// TIA Portal V17 export
// export: Created 2023-02-14T02:49:25.0894814Z, ExportSetting WithDefaults, DisplayName Totally Integrated Automation Portal, DisplayVersion V17, DisplayName TIA Portal Openness, DisplayVersion V17, DisplayName TIA Portal Teamcenter Gateway, DisplayVersion V17, DisplayName TIA Portal Version Control Interface, DisplayVersion V17, DisplayName SINAMICS Startdrive Advanced, DisplayVersion V17, DisplayName SINAMICS Startdrive G130, G150, S120, S150, SINAMICS MV, S210, DisplayVersion V17, DisplayName SINAMICS Startdrive G110M, G120, G120C, G120D, G120P, G115D, DisplayVersion V17, DisplayName STEP 7 Professional, DisplayVersion V17, DisplayName STEP 7 Safety, DisplayVersion V17, DisplayName WinCC Professional, DisplayVersion V17
FUNCTION_BLOCK "IO Analog Blending"   // FB10, LAD
{ S7_Optimized_Access := 'FALSE' }
VERSION : 0.1
// stored: AutoNumber true, IsIECCheckEnabled false, SetENOAutomatically false, UDAEnableTagReadback false
   VAR_INPUT
      Init : Bool;
      Reset : Bool;
   END_VAR
   VAR
      "LT-20.01" { S7_SetPoint := 'True'} : "Ana_w_K1K2";
      "LT-21.01" { S7_SetPoint := 'True'} : "Ana_w_K1K2";
      "LT-22.01" { S7_SetPoint := 'True'} : "Ana_w_K1K2";
      "LT-30.01" { S7_SetPoint := 'True'} : "Ana_w_K1K2";
      "LT-31.01" { S7_SetPoint := 'True'} : "Ana_w_K1K2";
      "LT-32.01" { S7_SetPoint := 'True'} : "Ana_w_K1K2";
      "FT-15.01" { S7_SetPoint := 'True'} : "Ana_w_K1K2";
      "FT-15.01Com" { S7_SetPoint := 'True'} : "Read FT Comm";
      "FT-22.01" { S7_SetPoint := 'True'} : "Ana_w_K1K2";
      "FT-22.01Com" { S7_SetPoint := 'True'} : "Read FT Comm";
      "FT-32.01" { S7_SetPoint := 'True'} : "Ana_w_K1K2";
      "FT-32.01Com" { S7_SetPoint := 'True'} : "Read FT Comm";
      "LT-40.01" { S7_SetPoint := 'True'} : "Ana_w_K1K2";
      "LT-41.01" { S7_SetPoint := 'True'} : "Ana_w_K1K2";
      "FT-00.01" { S7_SetPoint := 'True'} : "Ana_w_K1K2";
   END_VAR
BEGIN

REGION Network 1: LT-20.01
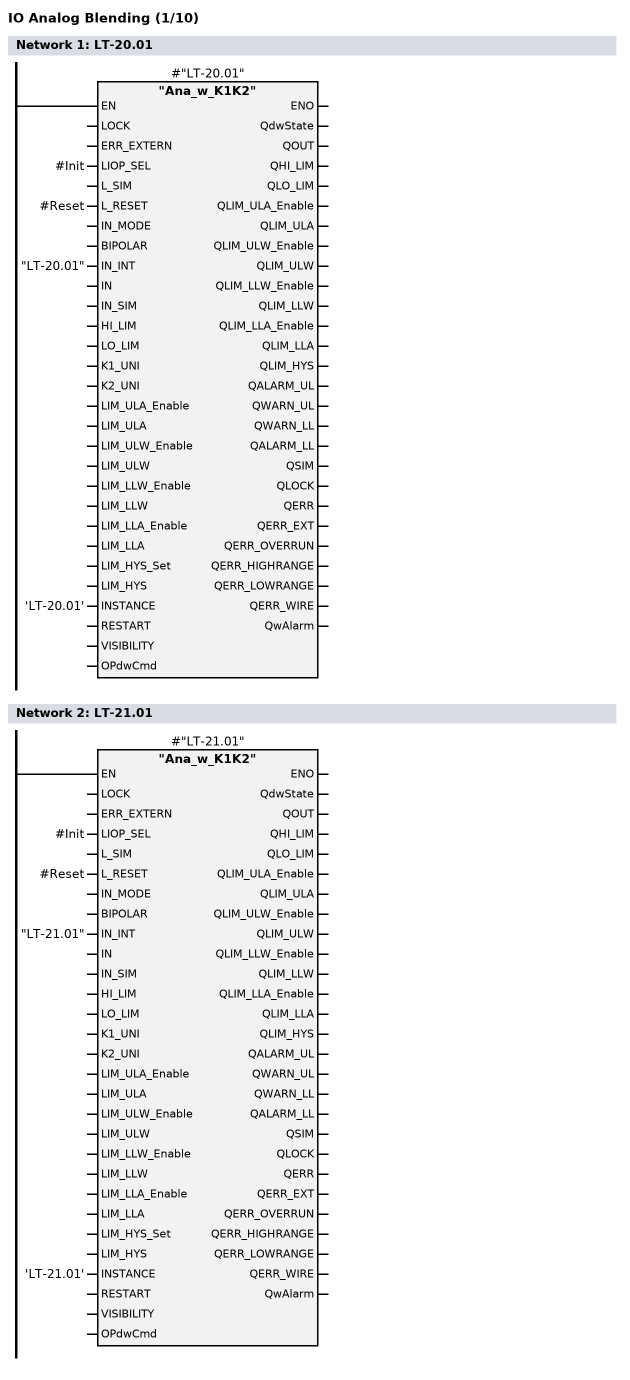
   RUNG wire#powerrail
      #"LT-20.01"(LOCK :=, ERR_EXTERN :=, LIOP_SEL := #Init, L_SIM :=, L_RESET := #Reset, IN_MODE :=, BIPOLAR :=, IN_INT := "LT-20.01", IN :=, IN_SIM :=, HI_LIM :=, LO_LIM :=, K1_UNI :=, K2_UNI :=, LIM_ULA_Enable :=, LIM_ULA :=, LIM_ULW_Enable :=, LIM_ULW :=, LIM_LLW_Enable :=, LIM_LLW :=, LIM_LLA_Enable :=, LIM_LLA :=, LIM_HYS_Set :=, LIM_HYS :=, INSTANCE := 'LT-20.01', RESTART :=, VISIBILITY :=, OPdwCmd :=, QdwState =>, QOUT =>, QHI_LIM =>, QLO_LIM =>, QLIM_ULA_Enable =>, QLIM_ULA =>, QLIM_ULW_Enable =>, QLIM_ULW =>, QLIM_LLW_Enable =>, QLIM_LLW =>, QLIM_LLA_Enable =>, QLIM_LLA =>, QLIM_HYS =>, QALARM_UL =>, QWARN_UL =>, QWARN_LL =>, QALARM_LL =>, QSIM =>, QLOCK =>, QERR =>, QERR_EXT =>, QERR_OVERRUN =>, QERR_HIGHRANGE =>, QERR_LOWRANGE =>, QERR_WIRE =>, QwAlarm =>)
   END_RUNG
   // the same network as SCL:
   #"LT-20.01"(LIOP_SEL := #Init, L_RESET := #Reset, IN_INT := "LT-20.01", INSTANCE := 'LT-20.01');   // "Ana_w_K1K2"
END_REGION

REGION Network 2: LT-21.01
   RUNG wire#powerrail
      #"LT-21.01"(LOCK :=, ERR_EXTERN :=, LIOP_SEL := #Init, L_SIM :=, L_RESET := #Reset, IN_MODE :=, BIPOLAR :=, IN_INT := "LT-21.01", IN :=, IN_SIM :=, HI_LIM :=, LO_LIM :=, K1_UNI :=, K2_UNI :=, LIM_ULA_Enable :=, LIM_ULA :=, LIM_ULW_Enable :=, LIM_ULW :=, LIM_LLW_Enable :=, LIM_LLW :=, LIM_LLA_Enable :=, LIM_LLA :=, LIM_HYS_Set :=, LIM_HYS :=, INSTANCE := 'LT-21.01', RESTART :=, VISIBILITY :=, OPdwCmd :=, QdwState =>, QOUT =>, QHI_LIM =>, QLO_LIM =>, QLIM_ULA_Enable =>, QLIM_ULA =>, QLIM_ULW_Enable =>, QLIM_ULW =>, QLIM_LLW_Enable =>, QLIM_LLW =>, QLIM_LLA_Enable =>, QLIM_LLA =>, QLIM_HYS =>, QALARM_UL =>, QWARN_UL =>, QWARN_LL =>, QALARM_LL =>, QSIM =>, QLOCK =>, QERR =>, QERR_EXT =>, QERR_OVERRUN =>, QERR_HIGHRANGE =>, QERR_LOWRANGE =>, QERR_WIRE =>, QwAlarm =>)
   END_RUNG
   // the same network as SCL:
   #"LT-21.01"(LIOP_SEL := #Init, L_RESET := #Reset, IN_INT := "LT-21.01", INSTANCE := 'LT-21.01');   // "Ana_w_K1K2"
END_REGION

REGION Network 3: LT-22.01
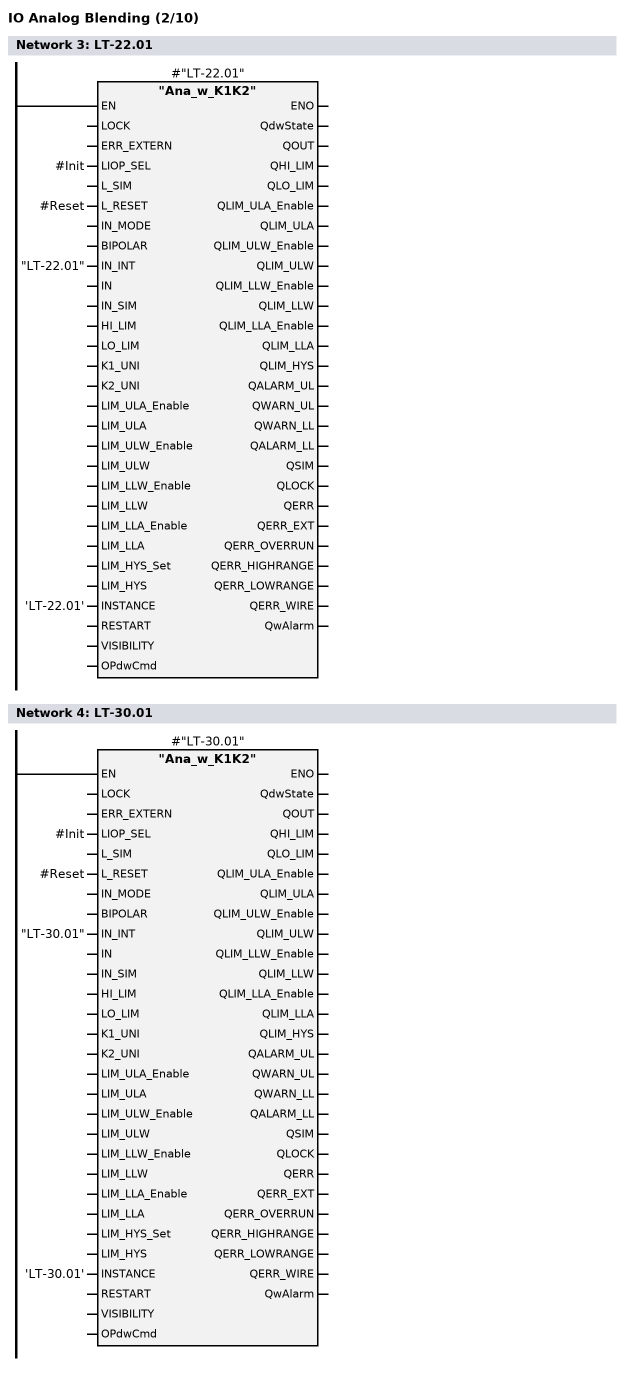
   RUNG wire#powerrail
      #"LT-22.01"(LOCK :=, ERR_EXTERN :=, LIOP_SEL := #Init, L_SIM :=, L_RESET := #Reset, IN_MODE :=, BIPOLAR :=, IN_INT := "LT-22.01", IN :=, IN_SIM :=, HI_LIM :=, LO_LIM :=, K1_UNI :=, K2_UNI :=, LIM_ULA_Enable :=, LIM_ULA :=, LIM_ULW_Enable :=, LIM_ULW :=, LIM_LLW_Enable :=, LIM_LLW :=, LIM_LLA_Enable :=, LIM_LLA :=, LIM_HYS_Set :=, LIM_HYS :=, INSTANCE := 'LT-22.01', RESTART :=, VISIBILITY :=, OPdwCmd :=, QdwState =>, QOUT =>, QHI_LIM =>, QLO_LIM =>, QLIM_ULA_Enable =>, QLIM_ULA =>, QLIM_ULW_Enable =>, QLIM_ULW =>, QLIM_LLW_Enable =>, QLIM_LLW =>, QLIM_LLA_Enable =>, QLIM_LLA =>, QLIM_HYS =>, QALARM_UL =>, QWARN_UL =>, QWARN_LL =>, QALARM_LL =>, QSIM =>, QLOCK =>, QERR =>, QERR_EXT =>, QERR_OVERRUN =>, QERR_HIGHRANGE =>, QERR_LOWRANGE =>, QERR_WIRE =>, QwAlarm =>)
   END_RUNG
   // the same network as SCL:
   #"LT-22.01"(LIOP_SEL := #Init, L_RESET := #Reset, IN_INT := "LT-22.01", INSTANCE := 'LT-22.01');   // "Ana_w_K1K2"
END_REGION

REGION Network 4: LT-30.01
   RUNG wire#powerrail
      #"LT-30.01"(LOCK :=, ERR_EXTERN :=, LIOP_SEL := #Init, L_SIM :=, L_RESET := #Reset, IN_MODE :=, BIPOLAR :=, IN_INT := "LT-30.01", IN :=, IN_SIM :=, HI_LIM :=, LO_LIM :=, K1_UNI :=, K2_UNI :=, LIM_ULA_Enable :=, LIM_ULA :=, LIM_ULW_Enable :=, LIM_ULW :=, LIM_LLW_Enable :=, LIM_LLW :=, LIM_LLA_Enable :=, LIM_LLA :=, LIM_HYS_Set :=, LIM_HYS :=, INSTANCE := 'LT-30.01', RESTART :=, VISIBILITY :=, OPdwCmd :=, QdwState =>, QOUT =>, QHI_LIM =>, QLO_LIM =>, QLIM_ULA_Enable =>, QLIM_ULA =>, QLIM_ULW_Enable =>, QLIM_ULW =>, QLIM_LLW_Enable =>, QLIM_LLW =>, QLIM_LLA_Enable =>, QLIM_LLA =>, QLIM_HYS =>, QALARM_UL =>, QWARN_UL =>, QWARN_LL =>, QALARM_LL =>, QSIM =>, QLOCK =>, QERR =>, QERR_EXT =>, QERR_OVERRUN =>, QERR_HIGHRANGE =>, QERR_LOWRANGE =>, QERR_WIRE =>, QwAlarm =>)
   END_RUNG
   // the same network as SCL:
   #"LT-30.01"(LIOP_SEL := #Init, L_RESET := #Reset, IN_INT := "LT-30.01", INSTANCE := 'LT-30.01');   // "Ana_w_K1K2"
END_REGION

REGION Network 5: LT-31.01
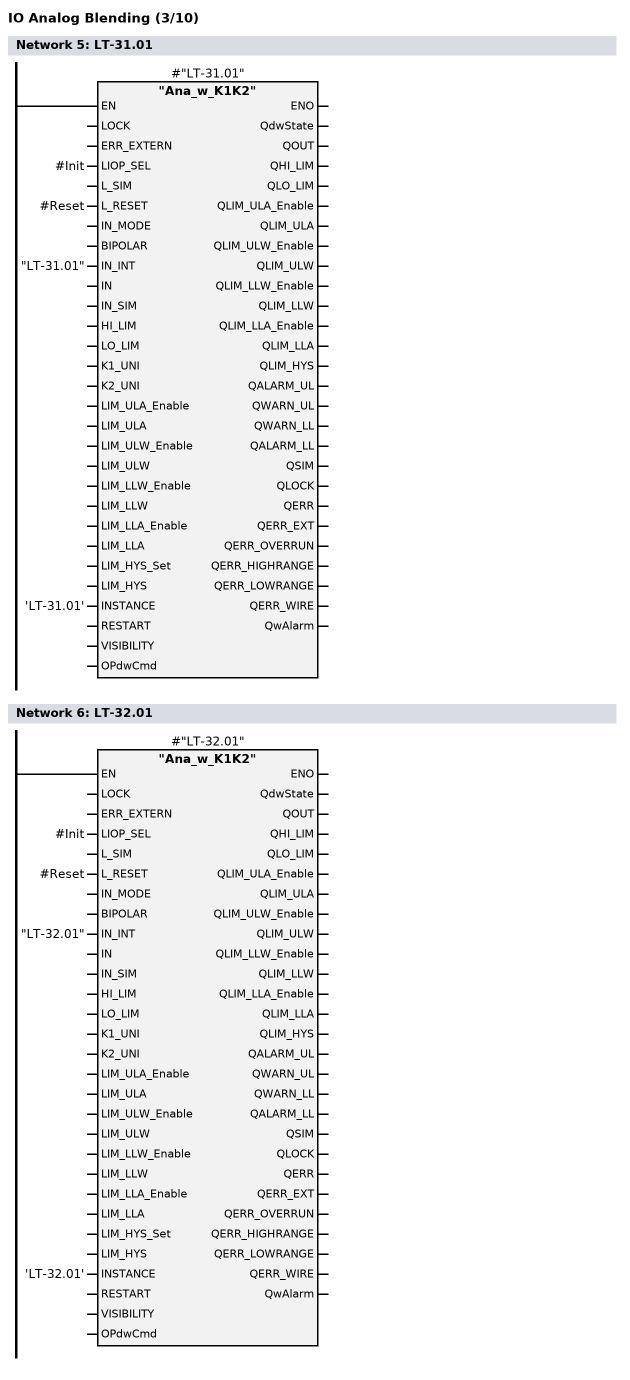
   RUNG wire#powerrail
      #"LT-31.01"(LOCK :=, ERR_EXTERN :=, LIOP_SEL := #Init, L_SIM :=, L_RESET := #Reset, IN_MODE :=, BIPOLAR :=, IN_INT := "LT-31.01", IN :=, IN_SIM :=, HI_LIM :=, LO_LIM :=, K1_UNI :=, K2_UNI :=, LIM_ULA_Enable :=, LIM_ULA :=, LIM_ULW_Enable :=, LIM_ULW :=, LIM_LLW_Enable :=, LIM_LLW :=, LIM_LLA_Enable :=, LIM_LLA :=, LIM_HYS_Set :=, LIM_HYS :=, INSTANCE := 'LT-31.01', RESTART :=, VISIBILITY :=, OPdwCmd :=, QdwState =>, QOUT =>, QHI_LIM =>, QLO_LIM =>, QLIM_ULA_Enable =>, QLIM_ULA =>, QLIM_ULW_Enable =>, QLIM_ULW =>, QLIM_LLW_Enable =>, QLIM_LLW =>, QLIM_LLA_Enable =>, QLIM_LLA =>, QLIM_HYS =>, QALARM_UL =>, QWARN_UL =>, QWARN_LL =>, QALARM_LL =>, QSIM =>, QLOCK =>, QERR =>, QERR_EXT =>, QERR_OVERRUN =>, QERR_HIGHRANGE =>, QERR_LOWRANGE =>, QERR_WIRE =>, QwAlarm =>)
   END_RUNG
   // the same network as SCL:
   #"LT-31.01"(LIOP_SEL := #Init, L_RESET := #Reset, IN_INT := "LT-31.01", INSTANCE := 'LT-31.01');   // "Ana_w_K1K2"
END_REGION

REGION Network 6: LT-32.01
   RUNG wire#powerrail
      #"LT-32.01"(LOCK :=, ERR_EXTERN :=, LIOP_SEL := #Init, L_SIM :=, L_RESET := #Reset, IN_MODE :=, BIPOLAR :=, IN_INT := "LT-32.01", IN :=, IN_SIM :=, HI_LIM :=, LO_LIM :=, K1_UNI :=, K2_UNI :=, LIM_ULA_Enable :=, LIM_ULA :=, LIM_ULW_Enable :=, LIM_ULW :=, LIM_LLW_Enable :=, LIM_LLW :=, LIM_LLA_Enable :=, LIM_LLA :=, LIM_HYS_Set :=, LIM_HYS :=, INSTANCE := 'LT-32.01', RESTART :=, VISIBILITY :=, OPdwCmd :=, QdwState =>, QOUT =>, QHI_LIM =>, QLO_LIM =>, QLIM_ULA_Enable =>, QLIM_ULA =>, QLIM_ULW_Enable =>, QLIM_ULW =>, QLIM_LLW_Enable =>, QLIM_LLW =>, QLIM_LLA_Enable =>, QLIM_LLA =>, QLIM_HYS =>, QALARM_UL =>, QWARN_UL =>, QWARN_LL =>, QALARM_LL =>, QSIM =>, QLOCK =>, QERR =>, QERR_EXT =>, QERR_OVERRUN =>, QERR_HIGHRANGE =>, QERR_LOWRANGE =>, QERR_WIRE =>, QwAlarm =>)
   END_RUNG
   // the same network as SCL:
   #"LT-32.01"(LIOP_SEL := #Init, L_RESET := #Reset, IN_INT := "LT-32.01", INSTANCE := 'LT-32.01');   // "Ana_w_K1K2"
END_REGION

REGION Network 7: LT-40.01
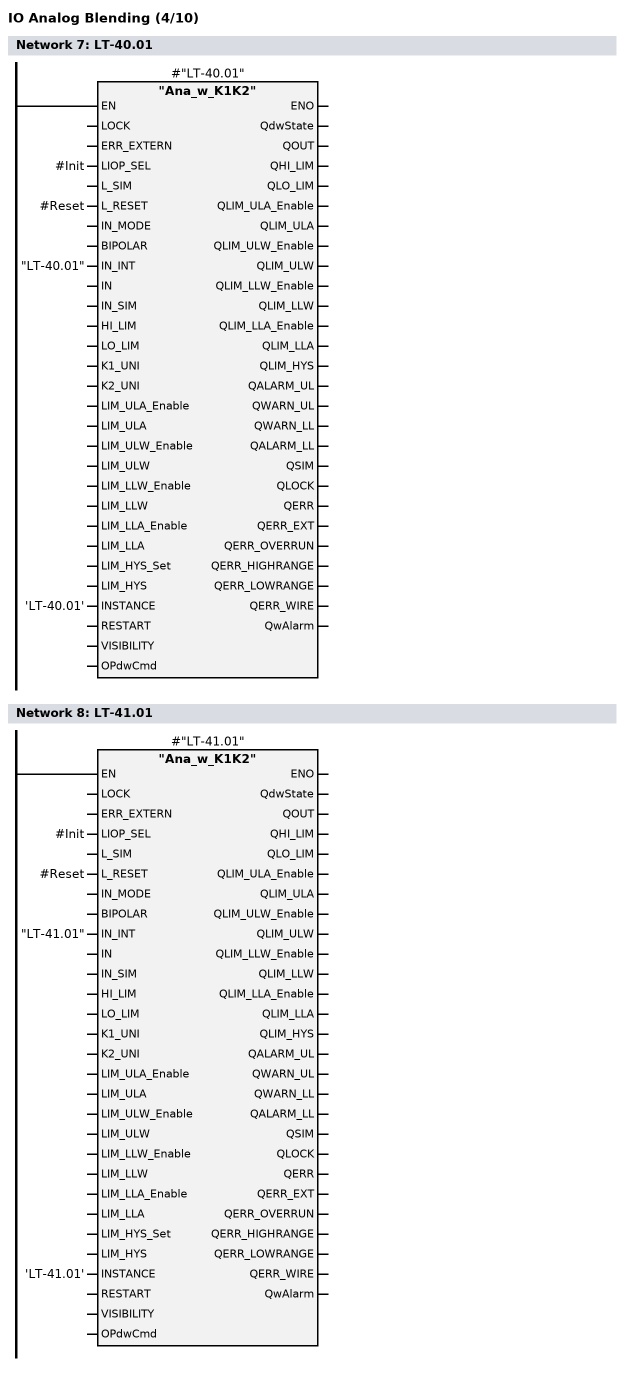
   RUNG wire#powerrail
      #"LT-40.01"(LOCK :=, ERR_EXTERN :=, LIOP_SEL := #Init, L_SIM :=, L_RESET := #Reset, IN_MODE :=, BIPOLAR :=, IN_INT := "LT-40.01", IN :=, IN_SIM :=, HI_LIM :=, LO_LIM :=, K1_UNI :=, K2_UNI :=, LIM_ULA_Enable :=, LIM_ULA :=, LIM_ULW_Enable :=, LIM_ULW :=, LIM_LLW_Enable :=, LIM_LLW :=, LIM_LLA_Enable :=, LIM_LLA :=, LIM_HYS_Set :=, LIM_HYS :=, INSTANCE := 'LT-40.01', RESTART :=, VISIBILITY :=, OPdwCmd :=, QdwState =>, QOUT =>, QHI_LIM =>, QLO_LIM =>, QLIM_ULA_Enable =>, QLIM_ULA =>, QLIM_ULW_Enable =>, QLIM_ULW =>, QLIM_LLW_Enable =>, QLIM_LLW =>, QLIM_LLA_Enable =>, QLIM_LLA =>, QLIM_HYS =>, QALARM_UL =>, QWARN_UL =>, QWARN_LL =>, QALARM_LL =>, QSIM =>, QLOCK =>, QERR =>, QERR_EXT =>, QERR_OVERRUN =>, QERR_HIGHRANGE =>, QERR_LOWRANGE =>, QERR_WIRE =>, QwAlarm =>)
   END_RUNG
   // the same network as SCL:
   #"LT-40.01"(LIOP_SEL := #Init, L_RESET := #Reset, IN_INT := "LT-40.01", INSTANCE := 'LT-40.01');   // "Ana_w_K1K2"
END_REGION

REGION Network 8: LT-41.01
   RUNG wire#powerrail
      #"LT-41.01"(LOCK :=, ERR_EXTERN :=, LIOP_SEL := #Init, L_SIM :=, L_RESET := #Reset, IN_MODE :=, BIPOLAR :=, IN_INT := "LT-41.01", IN :=, IN_SIM :=, HI_LIM :=, LO_LIM :=, K1_UNI :=, K2_UNI :=, LIM_ULA_Enable :=, LIM_ULA :=, LIM_ULW_Enable :=, LIM_ULW :=, LIM_LLW_Enable :=, LIM_LLW :=, LIM_LLA_Enable :=, LIM_LLA :=, LIM_HYS_Set :=, LIM_HYS :=, INSTANCE := 'LT-41.01', RESTART :=, VISIBILITY :=, OPdwCmd :=, QdwState =>, QOUT =>, QHI_LIM =>, QLO_LIM =>, QLIM_ULA_Enable =>, QLIM_ULA =>, QLIM_ULW_Enable =>, QLIM_ULW =>, QLIM_LLW_Enable =>, QLIM_LLW =>, QLIM_LLA_Enable =>, QLIM_LLA =>, QLIM_HYS =>, QALARM_UL =>, QWARN_UL =>, QWARN_LL =>, QALARM_LL =>, QSIM =>, QLOCK =>, QERR =>, QERR_EXT =>, QERR_OVERRUN =>, QERR_HIGHRANGE =>, QERR_LOWRANGE =>, QERR_WIRE =>, QwAlarm =>)
   END_RUNG
   // the same network as SCL:
   #"LT-41.01"(LIOP_SEL := #Init, L_RESET := #Reset, IN_INT := "LT-41.01", INSTANCE := 'LT-41.01');   // "Ana_w_K1K2"
END_REGION

REGION Network 9: FT-15.01 Communication
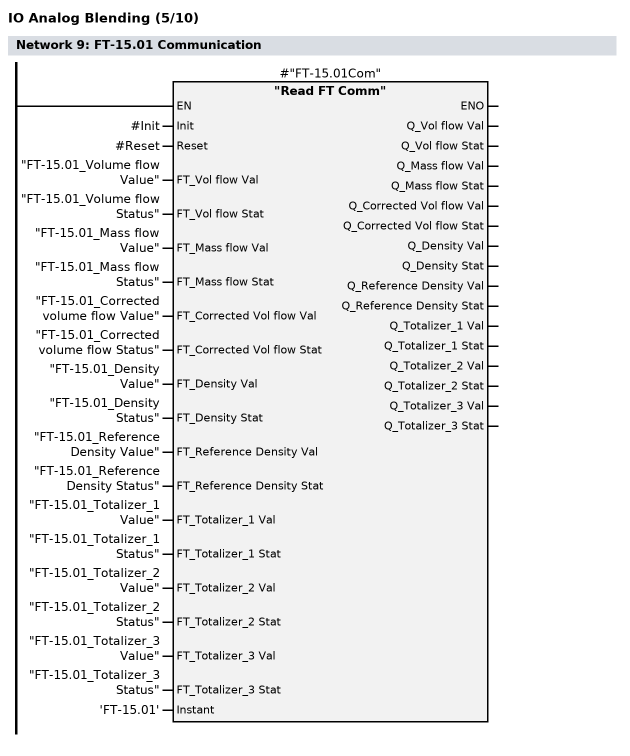
   RUNG wire#powerrail
      #"FT-15.01Com"(Init := #Init, Reset := #Reset, "FT_Vol flow Val" := "FT-15.01_Volume flow Value", "FT_Vol flow Stat" := "FT-15.01_Volume flow Status", "FT_Mass flow Val" := "FT-15.01_Mass flow Value", "FT_Mass flow Stat" := "FT-15.01_Mass flow Status", "FT_Corrected Vol flow Val" := "FT-15.01_Corrected volume flow Value", "FT_Corrected Vol flow Stat" := "FT-15.01_Corrected volume flow Status", "FT_Density Val" := "FT-15.01_Density Value", "FT_Density Stat" := "FT-15.01_Density Status", "FT_Reference Density Val" := "FT-15.01_Reference Density Value", "FT_Reference Density Stat" := "FT-15.01_Reference Density Status", "FT_Totalizer_1 Val" := "FT-15.01_Totalizer_1 Value", "FT_Totalizer_1 Stat" := "FT-15.01_Totalizer_1 Status", "FT_Totalizer_2 Val" := "FT-15.01_Totalizer_2 Value", "FT_Totalizer_2 Stat" := "FT-15.01_Totalizer_2 Status", "FT_Totalizer_3 Val" := "FT-15.01_Totalizer_3 Value", "FT_Totalizer_3 Stat" := "FT-15.01_Totalizer_3 Status", Instant := 'FT-15.01', "Q_Vol flow Val" =>, "Q_Vol flow Stat" =>, "Q_Mass flow Val" =>, "Q_Mass flow Stat" =>, "Q_Corrected Vol flow Val" =>, "Q_Corrected Vol flow Stat" =>, "Q_Density Val" =>, "Q_Density Stat" =>, "Q_Reference Density Val" =>, "Q_Reference Density Stat" =>, "Q_Totalizer_1 Val" =>, "Q_Totalizer_1 Stat" =>, "Q_Totalizer_2 Val" =>, "Q_Totalizer_2 Stat" =>, "Q_Totalizer_3 Val" =>, "Q_Totalizer_3 Stat" =>)
   END_RUNG
   // the same network as SCL:
   #"FT-15.01Com"(Init := #Init,   // "Read FT Comm"
                  Reset := #Reset,
                  "FT_Vol flow Val" := "FT-15.01_Volume flow Value",
                  "FT_Vol flow Stat" := "FT-15.01_Volume flow Status",
                  "FT_Mass flow Val" := "FT-15.01_Mass flow Value",
                  "FT_Mass flow Stat" := "FT-15.01_Mass flow Status",
                  "FT_Corrected Vol flow Val" := "FT-15.01_Corrected volume flow Value",
                  "FT_Corrected Vol flow Stat" := "FT-15.01_Corrected volume flow Status",
                  "FT_Density Val" := "FT-15.01_Density Value",
                  "FT_Density Stat" := "FT-15.01_Density Status",
                  "FT_Reference Density Val" := "FT-15.01_Reference Density Value",
                  "FT_Reference Density Stat" := "FT-15.01_Reference Density Status",
                  "FT_Totalizer_1 Val" := "FT-15.01_Totalizer_1 Value",
                  "FT_Totalizer_1 Stat" := "FT-15.01_Totalizer_1 Status",
                  "FT_Totalizer_2 Val" := "FT-15.01_Totalizer_2 Value",
                  "FT_Totalizer_2 Stat" := "FT-15.01_Totalizer_2 Status",
                  "FT_Totalizer_3 Val" := "FT-15.01_Totalizer_3 Value",
                  "FT_Totalizer_3 Stat" := "FT-15.01_Totalizer_3 Status",
                  Instant := 'FT-15.01');
END_REGION

REGION Network 10: FT-15.01 Flowrate
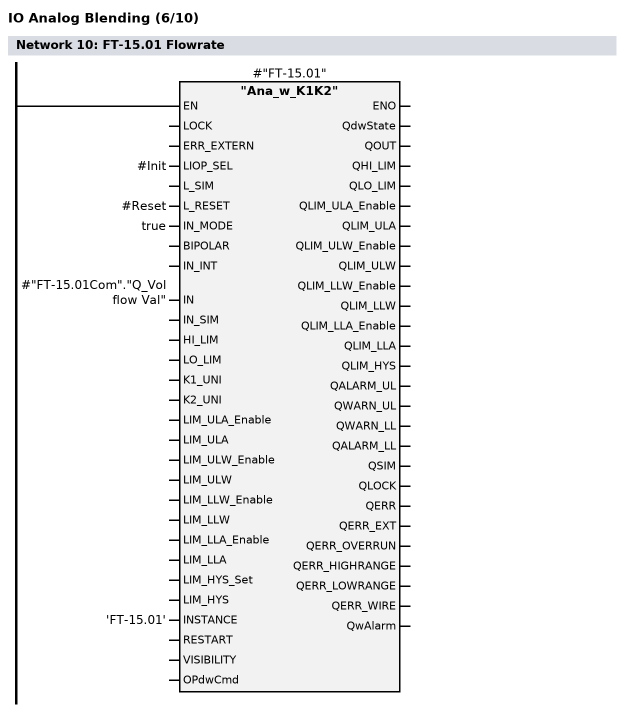
   RUNG wire#powerrail
      #"FT-15.01"(LOCK :=, ERR_EXTERN :=, LIOP_SEL := #Init, L_SIM :=, L_RESET := #Reset, IN_MODE := true, BIPOLAR :=, IN_INT :=, IN := #"FT-15.01Com"."Q_Vol flow Val", IN_SIM :=, HI_LIM :=, LO_LIM :=, K1_UNI :=, K2_UNI :=, LIM_ULA_Enable :=, LIM_ULA :=, LIM_ULW_Enable :=, LIM_ULW :=, LIM_LLW_Enable :=, LIM_LLW :=, LIM_LLA_Enable :=, LIM_LLA :=, LIM_HYS_Set :=, LIM_HYS :=, INSTANCE := 'FT-15.01', RESTART :=, VISIBILITY :=, OPdwCmd :=, QdwState =>, QOUT =>, QHI_LIM =>, QLO_LIM =>, QLIM_ULA_Enable =>, QLIM_ULA =>, QLIM_ULW_Enable =>, QLIM_ULW =>, QLIM_LLW_Enable =>, QLIM_LLW =>, QLIM_LLA_Enable =>, QLIM_LLA =>, QLIM_HYS =>, QALARM_UL =>, QWARN_UL =>, QWARN_LL =>, QALARM_LL =>, QSIM =>, QLOCK =>, QERR =>, QERR_EXT =>, QERR_OVERRUN =>, QERR_HIGHRANGE =>, QERR_LOWRANGE =>, QERR_WIRE =>, QwAlarm =>)
   END_RUNG
   // the same network as SCL:
   #"FT-15.01"(LIOP_SEL := #Init,   // "Ana_w_K1K2"
               L_RESET := #Reset,
               IN_MODE := true,
               IN := #"FT-15.01Com"."Q_Vol flow Val",
               INSTANCE := 'FT-15.01');
END_REGION

REGION Network 11: FT-22.01 Communication
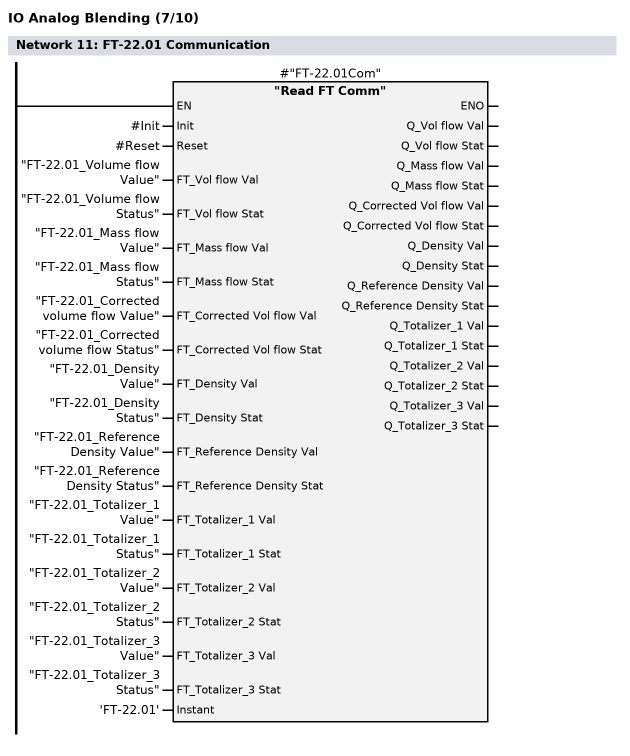
   RUNG wire#powerrail
      #"FT-22.01Com"(Init := #Init, Reset := #Reset, "FT_Vol flow Val" := "FT-22.01_Volume flow Value", "FT_Vol flow Stat" := "FT-22.01_Volume flow Status", "FT_Mass flow Val" := "FT-22.01_Mass flow Value", "FT_Mass flow Stat" := "FT-22.01_Mass flow Status", "FT_Corrected Vol flow Val" := "FT-22.01_Corrected volume flow Value", "FT_Corrected Vol flow Stat" := "FT-22.01_Corrected volume flow Status", "FT_Density Val" := "FT-22.01_Density Value", "FT_Density Stat" := "FT-22.01_Density Status", "FT_Reference Density Val" := "FT-22.01_Reference Density Value", "FT_Reference Density Stat" := "FT-22.01_Reference Density Status", "FT_Totalizer_1 Val" := "FT-22.01_Totalizer_1 Value", "FT_Totalizer_1 Stat" := "FT-22.01_Totalizer_1 Status", "FT_Totalizer_2 Val" := "FT-22.01_Totalizer_2 Value", "FT_Totalizer_2 Stat" := "FT-22.01_Totalizer_2 Status", "FT_Totalizer_3 Val" := "FT-22.01_Totalizer_3 Value", "FT_Totalizer_3 Stat" := "FT-22.01_Totalizer_3 Status", Instant := 'FT-22.01', "Q_Vol flow Val" =>, "Q_Vol flow Stat" =>, "Q_Mass flow Val" =>, "Q_Mass flow Stat" =>, "Q_Corrected Vol flow Val" =>, "Q_Corrected Vol flow Stat" =>, "Q_Density Val" =>, "Q_Density Stat" =>, "Q_Reference Density Val" =>, "Q_Reference Density Stat" =>, "Q_Totalizer_1 Val" =>, "Q_Totalizer_1 Stat" =>, "Q_Totalizer_2 Val" =>, "Q_Totalizer_2 Stat" =>, "Q_Totalizer_3 Val" =>, "Q_Totalizer_3 Stat" =>)
   END_RUNG
   // the same network as SCL:
   #"FT-22.01Com"(Init := #Init,   // "Read FT Comm"
                  Reset := #Reset,
                  "FT_Vol flow Val" := "FT-22.01_Volume flow Value",
                  "FT_Vol flow Stat" := "FT-22.01_Volume flow Status",
                  "FT_Mass flow Val" := "FT-22.01_Mass flow Value",
                  "FT_Mass flow Stat" := "FT-22.01_Mass flow Status",
                  "FT_Corrected Vol flow Val" := "FT-22.01_Corrected volume flow Value",
                  "FT_Corrected Vol flow Stat" := "FT-22.01_Corrected volume flow Status",
                  "FT_Density Val" := "FT-22.01_Density Value",
                  "FT_Density Stat" := "FT-22.01_Density Status",
                  "FT_Reference Density Val" := "FT-22.01_Reference Density Value",
                  "FT_Reference Density Stat" := "FT-22.01_Reference Density Status",
                  "FT_Totalizer_1 Val" := "FT-22.01_Totalizer_1 Value",
                  "FT_Totalizer_1 Stat" := "FT-22.01_Totalizer_1 Status",
                  "FT_Totalizer_2 Val" := "FT-22.01_Totalizer_2 Value",
                  "FT_Totalizer_2 Stat" := "FT-22.01_Totalizer_2 Status",
                  "FT_Totalizer_3 Val" := "FT-22.01_Totalizer_3 Value",
                  "FT_Totalizer_3 Stat" := "FT-22.01_Totalizer_3 Status",
                  Instant := 'FT-22.01');
END_REGION

REGION Network 12: FT-22.01 Flowrate
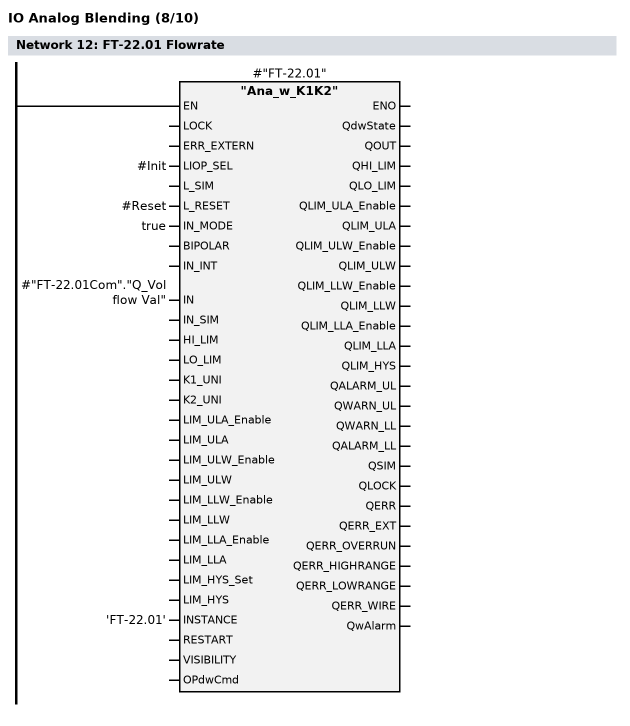
   RUNG wire#powerrail
      #"FT-22.01"(LOCK :=, ERR_EXTERN :=, LIOP_SEL := #Init, L_SIM :=, L_RESET := #Reset, IN_MODE := true, BIPOLAR :=, IN_INT :=, IN := #"FT-22.01Com"."Q_Vol flow Val", IN_SIM :=, HI_LIM :=, LO_LIM :=, K1_UNI :=, K2_UNI :=, LIM_ULA_Enable :=, LIM_ULA :=, LIM_ULW_Enable :=, LIM_ULW :=, LIM_LLW_Enable :=, LIM_LLW :=, LIM_LLA_Enable :=, LIM_LLA :=, LIM_HYS_Set :=, LIM_HYS :=, INSTANCE := 'FT-22.01', RESTART :=, VISIBILITY :=, OPdwCmd :=, QdwState =>, QOUT =>, QHI_LIM =>, QLO_LIM =>, QLIM_ULA_Enable =>, QLIM_ULA =>, QLIM_ULW_Enable =>, QLIM_ULW =>, QLIM_LLW_Enable =>, QLIM_LLW =>, QLIM_LLA_Enable =>, QLIM_LLA =>, QLIM_HYS =>, QALARM_UL =>, QWARN_UL =>, QWARN_LL =>, QALARM_LL =>, QSIM =>, QLOCK =>, QERR =>, QERR_EXT =>, QERR_OVERRUN =>, QERR_HIGHRANGE =>, QERR_LOWRANGE =>, QERR_WIRE =>, QwAlarm =>)
   END_RUNG
   // the same network as SCL:
   #"FT-22.01"(LIOP_SEL := #Init,   // "Ana_w_K1K2"
               L_RESET := #Reset,
               IN_MODE := true,
               IN := #"FT-22.01Com"."Q_Vol flow Val",
               INSTANCE := 'FT-22.01');
END_REGION

REGION Network 13: FT-32.01 Communication
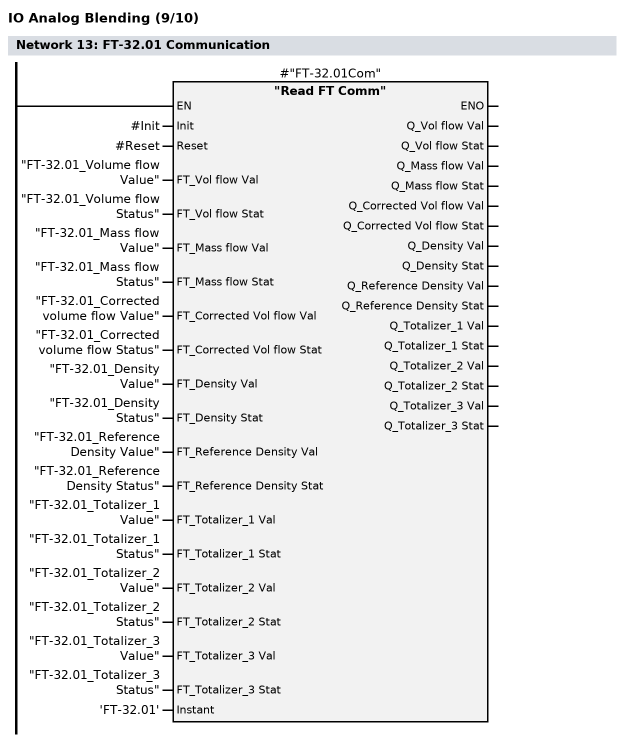
   RUNG wire#powerrail
      #"FT-32.01Com"(Init := #Init, Reset := #Reset, "FT_Vol flow Val" := "FT-32.01_Volume flow Value", "FT_Vol flow Stat" := "FT-32.01_Volume flow Status", "FT_Mass flow Val" := "FT-32.01_Mass flow Value", "FT_Mass flow Stat" := "FT-32.01_Mass flow Status", "FT_Corrected Vol flow Val" := "FT-32.01_Corrected volume flow Value", "FT_Corrected Vol flow Stat" := "FT-32.01_Corrected volume flow Status", "FT_Density Val" := "FT-32.01_Density Value", "FT_Density Stat" := "FT-32.01_Density Status", "FT_Reference Density Val" := "FT-32.01_Reference Density Value", "FT_Reference Density Stat" := "FT-32.01_Reference Density Status", "FT_Totalizer_1 Val" := "FT-32.01_Totalizer_1 Value", "FT_Totalizer_1 Stat" := "FT-32.01_Totalizer_1 Status", "FT_Totalizer_2 Val" := "FT-32.01_Totalizer_2 Value", "FT_Totalizer_2 Stat" := "FT-32.01_Totalizer_2 Status", "FT_Totalizer_3 Val" := "FT-32.01_Totalizer_3 Value", "FT_Totalizer_3 Stat" := "FT-32.01_Totalizer_3 Status", Instant := 'FT-32.01', "Q_Vol flow Val" =>, "Q_Vol flow Stat" =>, "Q_Mass flow Val" =>, "Q_Mass flow Stat" =>, "Q_Corrected Vol flow Val" =>, "Q_Corrected Vol flow Stat" =>, "Q_Density Val" =>, "Q_Density Stat" =>, "Q_Reference Density Val" =>, "Q_Reference Density Stat" =>, "Q_Totalizer_1 Val" =>, "Q_Totalizer_1 Stat" =>, "Q_Totalizer_2 Val" =>, "Q_Totalizer_2 Stat" =>, "Q_Totalizer_3 Val" =>, "Q_Totalizer_3 Stat" =>)
   END_RUNG
   // the same network as SCL:
   #"FT-32.01Com"(Init := #Init,   // "Read FT Comm"
                  Reset := #Reset,
                  "FT_Vol flow Val" := "FT-32.01_Volume flow Value",
                  "FT_Vol flow Stat" := "FT-32.01_Volume flow Status",
                  "FT_Mass flow Val" := "FT-32.01_Mass flow Value",
                  "FT_Mass flow Stat" := "FT-32.01_Mass flow Status",
                  "FT_Corrected Vol flow Val" := "FT-32.01_Corrected volume flow Value",
                  "FT_Corrected Vol flow Stat" := "FT-32.01_Corrected volume flow Status",
                  "FT_Density Val" := "FT-32.01_Density Value",
                  "FT_Density Stat" := "FT-32.01_Density Status",
                  "FT_Reference Density Val" := "FT-32.01_Reference Density Value",
                  "FT_Reference Density Stat" := "FT-32.01_Reference Density Status",
                  "FT_Totalizer_1 Val" := "FT-32.01_Totalizer_1 Value",
                  "FT_Totalizer_1 Stat" := "FT-32.01_Totalizer_1 Status",
                  "FT_Totalizer_2 Val" := "FT-32.01_Totalizer_2 Value",
                  "FT_Totalizer_2 Stat" := "FT-32.01_Totalizer_2 Status",
                  "FT_Totalizer_3 Val" := "FT-32.01_Totalizer_3 Value",
                  "FT_Totalizer_3 Stat" := "FT-32.01_Totalizer_3 Status",
                  Instant := 'FT-32.01');
END_REGION

REGION Network 14: FT-32.01 Flowrate
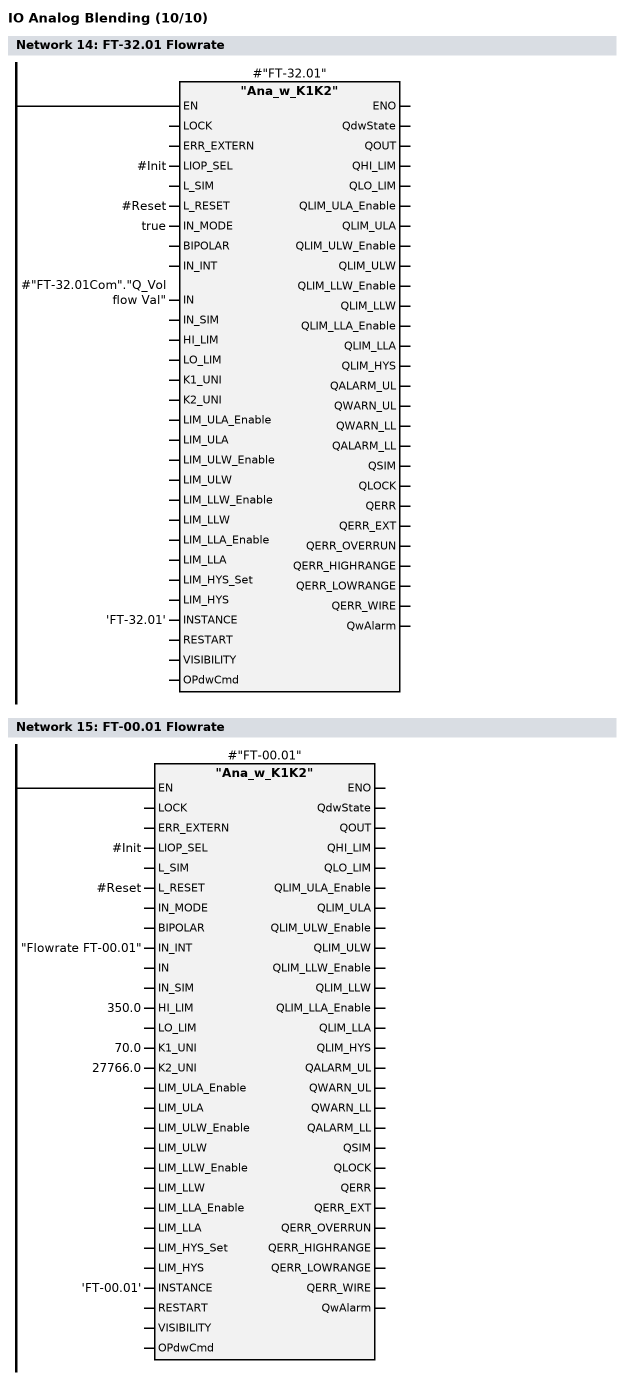
   RUNG wire#powerrail
      #"FT-32.01"(LOCK :=, ERR_EXTERN :=, LIOP_SEL := #Init, L_SIM :=, L_RESET := #Reset, IN_MODE := true, BIPOLAR :=, IN_INT :=, IN := #"FT-32.01Com"."Q_Vol flow Val", IN_SIM :=, HI_LIM :=, LO_LIM :=, K1_UNI :=, K2_UNI :=, LIM_ULA_Enable :=, LIM_ULA :=, LIM_ULW_Enable :=, LIM_ULW :=, LIM_LLW_Enable :=, LIM_LLW :=, LIM_LLA_Enable :=, LIM_LLA :=, LIM_HYS_Set :=, LIM_HYS :=, INSTANCE := 'FT-32.01', RESTART :=, VISIBILITY :=, OPdwCmd :=, QdwState =>, QOUT =>, QHI_LIM =>, QLO_LIM =>, QLIM_ULA_Enable =>, QLIM_ULA =>, QLIM_ULW_Enable =>, QLIM_ULW =>, QLIM_LLW_Enable =>, QLIM_LLW =>, QLIM_LLA_Enable =>, QLIM_LLA =>, QLIM_HYS =>, QALARM_UL =>, QWARN_UL =>, QWARN_LL =>, QALARM_LL =>, QSIM =>, QLOCK =>, QERR =>, QERR_EXT =>, QERR_OVERRUN =>, QERR_HIGHRANGE =>, QERR_LOWRANGE =>, QERR_WIRE =>, QwAlarm =>)
   END_RUNG
   // the same network as SCL:
   #"FT-32.01"(LIOP_SEL := #Init,   // "Ana_w_K1K2"
               L_RESET := #Reset,
               IN_MODE := true,
               IN := #"FT-32.01Com"."Q_Vol flow Val",
               INSTANCE := 'FT-32.01');
END_REGION

REGION Network 15: FT-00.01 Flowrate
   RUNG wire#powerrail
      #"FT-00.01"(LOCK :=, ERR_EXTERN :=, LIOP_SEL := #Init, L_SIM :=, L_RESET := #Reset, IN_MODE :=, BIPOLAR :=, IN_INT := "Flowrate FT-00.01", IN :=, IN_SIM :=, HI_LIM := 350.0, LO_LIM :=, K1_UNI := 70.0, K2_UNI := 27766.0, LIM_ULA_Enable :=, LIM_ULA :=, LIM_ULW_Enable :=, LIM_ULW :=, LIM_LLW_Enable :=, LIM_LLW :=, LIM_LLA_Enable :=, LIM_LLA :=, LIM_HYS_Set :=, LIM_HYS :=, INSTANCE := 'FT-00.01', RESTART :=, VISIBILITY :=, OPdwCmd :=, QdwState =>, QOUT =>, QHI_LIM =>, QLO_LIM =>, QLIM_ULA_Enable =>, QLIM_ULA =>, QLIM_ULW_Enable =>, QLIM_ULW =>, QLIM_LLW_Enable =>, QLIM_LLW =>, QLIM_LLA_Enable =>, QLIM_LLA =>, QLIM_HYS =>, QALARM_UL =>, QWARN_UL =>, QWARN_LL =>, QALARM_LL =>, QSIM =>, QLOCK =>, QERR =>, QERR_EXT =>, QERR_OVERRUN =>, QERR_HIGHRANGE =>, QERR_LOWRANGE =>, QERR_WIRE =>, QwAlarm =>)
   END_RUNG
   // the same network as SCL:
   #"FT-00.01"(LIOP_SEL := #Init,   // "Ana_w_K1K2"
               L_RESET := #Reset,
               IN_INT := "Flowrate FT-00.01",
               HI_LIM := 350.0,
               K1_UNI := 70.0,
               K2_UNI := 27766.0,
               INSTANCE := 'FT-00.01');
END_REGION
END_FUNCTION_BLOCK
